Staubli VAL3: readErrorTable.pgx

program readErrorTable(num errorNum_, string& msgTable_[], string& msg_[])
begin
  // get error message of the last cognex command from error message table
  errorNum_=abs(errorNum_)
  if (errorNum_>=0) and (errorNum_<size(msgTable_))
    msg_=msgTable_[errorNum_]
    if len(msg_)<2
      msg_="Unknown error"
    endIf
  else
    msg_="Unknown error"
  endIf
end
